TYPE ST_GUI_HMI :
STRUCT
END_STRUCT
END_TYPE

(* stored: Version 1.1.0.1, ProductVersion 3.1.4022.11
   DUT ST_GUI_HMI: Id {f634e8ff-154a-4be8-affd-2c46a10af667} *)
